Universal Robots PolyScope program: IAC009 PickFromTable.urp

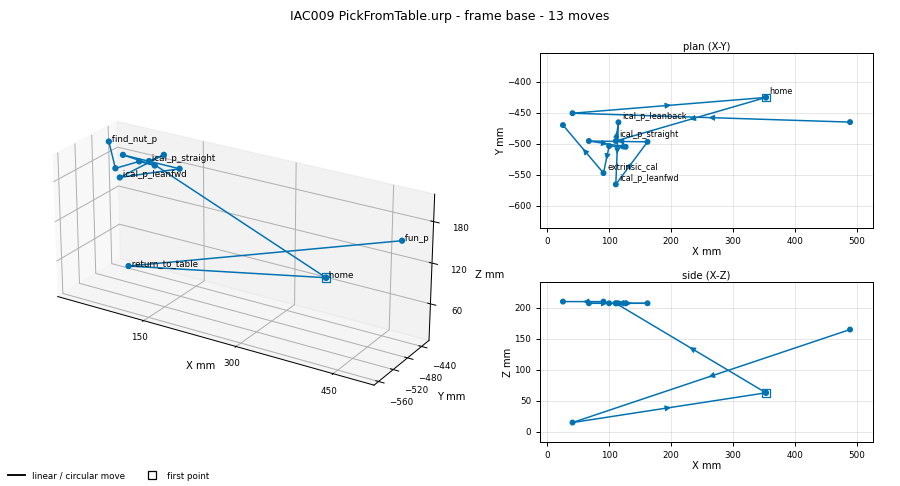
[picture p0: tool path of IAC009 PickFromTable.urp in frame base, 13 of 15 moves have a stored position in this frame; points joined in program order, loops and branches not executed]
Program IAC009 PickFromTable (installation=default directory=/programs createdIn=5.9.1.1031110 lastSavedIn=5.9.1.1031110 robotSerialNumber=20195501059)
Calibrated DH parameters: a=[0.000146, -0.418764, -0.053981, 0.000058, -0.000023, 0]; d=[0.162545, 37.319448, -206.067439, 168.881546, 0.09955, 0.099464]; alpha=[1.57004, -0.001979, 0.002304, 1.570607, -1.57066, 0]; deltaTheta=[0, -0.174616, -1.258233, 1.432844, -0.000001, 0]
BeforeStart
  URCap Gripper Activate (Robotiq_Grippers, Robotiq Inc.) dataModel(ResetAndActivateKey=false)
  initial_p := get_actual_tcp_pose()
  MoveJ speed 60 deg/s, acceleration 80 deg/s^2 (useActiveTCP=true) feature=Base
    Waypoint Waypoint (Variable): variable=initial_p
Robot Program (runOnlyOnce=true)
  URCap Gripper (Robotiq_Grippers, Robotiq Inc.) dataModel(position=100.0, force=100.0, speed=100.0, positionInDouble=100.0, forceInDouble=100.0, speedInDouble=100.0, slaveIds=[9], blocking=true)
  MoveL speed 250 mm/s, acceleration 1200 mm/s^2 (useActiveTCP=true) feature=Base
    Waypoint home: TCP in base x=353.458 y=-425.055 z=62.619 mm, rx=2.1827 ry=2.2595 rz=0 rad; joints [115.739, -73.375, 109.924, -126.542, 270.036, 113.788] deg; TCP offset x=0 y=0 z=174 mm, rx=0 ry=0 rz=0 rad
  Call vision_connect
  'Perform intrinsic calibration'
  MoveL speed 250 mm/s, acceleration 1200 mm/s^2 (useActiveTCP=true) feature=Base
    Waypoint ical_p_straight: TCP in base x=110.855 y=-495.374 z=207.252 mm, rx=1.1672 ry=2.7546 rz=-0.3884 rad; joints [86.306, -96.835, 118.195, -127.67, 271.92, 42.519] deg
    Call vis_start_intrinsic_cal
    Call vis_add_intrinsic_cal
    Waypoint ical_p_leanback: TCP in base x=115.098 y=-465.185 z=207.229 mm, rx=1.1297 ry=2.6702 rz=-0.5869 rad; joints [86.277, -104.564, 128.82, -139.297, 272.475, 42.708] deg
    Call vis_add_intrinsic_cal
    Waypoint ical_p_leanfwd: TCP in base x=110.84 y=-565.556 z=207.246 mm, rx=-1.2223 ry=-2.8743 rz=-0.1161 rad; joints [87.366, -76.554, 89.607, -98.733, 270.622, 43.42] deg
    Call vis_add_intrinsic_cal
    Waypoint ical_p_leanleft: TCP in base x=162.06 y=-496.773 z=207.271 mm, rx=-1.1054 ry=-2.7561 rz=0.5383 rad; joints [102.299, -90.049, 112.41, -125.743, 252.778, 53.986] deg
    Call vis_add_intrinsic_cal
    Waypoint ical_p_leanrgt: TCP in base x=67.326 y=-495.405 z=207.256 mm, rx=1.1363 ry=2.5701 rz=-0.2417 rad; joints [72.375, -99.02, 119.959, -122.988, 287.189, 31.913] deg
    Call vis_add_intrinsic_cal
    Waypoint ical_p_rotcw: TCP in base x=126.741 y=-504.81 z=207.25 mm, rx=1.7476 ry=2.492 rz=-0.4265 rad; joints [92.768, -92.929, 114.348, -126.478, 263.442, 71.995] deg
    Call vis_add_intrinsic_cal
    Waypoint ical_p_rotccw: TCP in base x=100.084 y=-503.616 z=207.257 mm, rx=0.6791 ry=2.8759 rz=-0.3469 rad; joints [81.53, -96.237, 117.124, -125.095, 278.363, 19.156] deg
    Call vis_add_intrinsic_cal
    Call vis_finish_intrinsic_cal
  'Perform extrinsic calibration'
  MoveL speed 250 mm/s, acceleration 1200 mm/s^2 (useActiveTCP=true) feature=Base
    Waypoint extrinsic_cal: TCP in base x=90.921 y=-547.266 z=209.993 mm, rx=2.2391 ry=2.2034 rz=0.0001 rad; joints [85.482, -81.971, 96.737, -104.753, 270.015, 86.406] deg
    Call vis_extrinsic_cal
  Call vis_load_pattern
  'Loop finding nut, pick, and replace in slightly random position until not DIN[1]'
  Loop While (checkContinuously=false) expression=digital_in[1]
    MoveL speed 250 mm/s, acceleration 1200 mm/s^2 (useActiveTCP=true) feature=Base
      Waypoint find_nut_p: TCP in base x=25.479 y=-469.683 z=209.989 mm, rx=-2.2392 ry=-2.2035 rz=-0.0001 rad; joints [76.599, -93.658, 108.914, -105.242, 270.035, 77.521] deg
      Call vis_find_pattern
      If norm(VFoundDx)≠999
        Script file /programs/IAC009 Adjust Position Script.script
          | cur_p = get_actual_tcp_pose()
          | cur_p[0] = cur_p[0] - VFoundDx
          | cur_p[1] = cur_p[1] + VFoundDy
          | movel(cur_p)
        Call vis_find_pattern
        MoveL speed 250 mm/s, acceleration 1200 mm/s^2 (useActiveTCP=true) feature=Base
          Waypoint VisToPickOffset (Relative): relativeFromPosition TCP in base x=22.407 y=-468.277 z=209.791 mm, rx=-2.239 ry=-2.2034 rz=-0.0006 rad; joints [76.178, -93.861, 109.126, -105.229, 270.035, 77.096] deg; TCP in base x=42.13 y=-449.159 z=14.069 mm, rx=-2.239 ry=-2.2034 rz=-0.0007 rad; joints [78.116, -80.323, 128.804, -138.442, 270.071, 79.085] deg
          Call pick
          Waypoint fun_p: TCP in base x=489.287 y=-464.869 z=164.848 mm, rx=1.7021 ry=1.563 rz=1.087 rad; joints [103.294, -67.911, 111.993, -144.657, 329.453, 114.262] deg
          Waypoint return_to_table: TCP in base x=40.885 y=-450.517 z=14.571 mm, rx=-2.7252 ry=-1.563 rz=0 rad; joints [77.993, -80.248, 128.607, -138.349, 270.067, 108.373] deg
          Script file /programs/IAC009 Place Random Script.script
            | cur_p = get_actual_tcp_pose()
            | cur_p[0] = cur_p[0] + (random() - 0.5) * 0.015
            | cur_p[1] = cur_p[1] + (random() - 0.5) * 0.015
            | movel(cur_p)
          Call place
  MoveL speed 250 mm/s, acceleration 1200 mm/s^2 (useActiveTCP=true) feature=Base
    Waypoint home: TCP in base x=353.458 y=-425.055 z=62.619 mm, rx=2.1827 ry=2.2595 rz=0 rad; joints [115.739, -73.375, 109.924, -126.542, 270.036, 113.788] deg
  Call vision_disconnect
SubProgram  [hidden by the author, left out]
SubProgram  [hidden by the author, left out]
SubProgram  [hidden by the author, left out]
SubProgram  [hidden by the author, left out]
SubProgram vision_acquire_only [hidden by the author, left out]
SubProgram  [hidden by the author, left out]
SubProgram  [hidden by the author, left out]
SubProgram  [hidden by the author, left out]
SubProgram  [hidden by the author, left out]
SubProgram  [hidden by the author, left out]
SubProgram  [hidden by the author, left out]
SubProgram vision_connect [hidden by the author, left out]
SubProgram vis_start_intrinsic_cal [hidden by the author, left out]
SubProgram vis_add_intrinsic_cal [hidden by the author, left out]
SubProgram vis_finish_intrinsic_cal [hidden by the author, left out]
SubProgram vis_extrinsic_cal [hidden by the author, left out]
SubProgram vis_load_pattern [hidden by the author, left out]
SubProgram vis_find_pattern [hidden by the author, left out]
SubProgram pick [hidden by the author, left out]
SubProgram place [hidden by the author, left out]
SubProgram vision_disconnect [hidden by the author, left out]
